FUNCTION_BLOCK PUBLIC AutomaticControl
VAR_INPUT
	Switch: BOOL;
END_VAR
VAR
	ExecutingRecipe1: BOOL := FALSE;
	ExecutingRecipe2: BOOL := FALSE;
	SwitchedManualAuto: BOOL := FALSE;
	initialized: BOOL := FALSE;
	State: INT := 0;
END_VAR
VAR_OUTPUT
	Output: BOOL;
END_VAR

// Initially go to position (0,0,0,0) and initialize motors
IF NOT IO.Initialized THEN
	Initialize();
ELSE
	//Safety();	// to stop when out of range
	
	// COUNTING (POSITION):
	CountPosition();	// FOR MANUAL MODE
	
	// RESET THE POSITION:
	(*IF (Automatic.RotationPositionAuto - Automatic.RotationPositionCurrent > 20 OR Automatic.RotationPositionAuto - Automatic.RotationPositionCurrent > 20) AND IO.SwitchedToAutomatic THEN
		IF Automatic.RotationPositionAuto - Automatic.RotationPositionCurrent > 20 THEN
			IO.MotorRotationDirection := 0;
		ELSE
			IO.MotorRotationDirection := 1;
		END_IF
		IO.MotorRotation := 1;
	ELSE 
		IO.MotorRotation := 0;
		IO.SwitchedToAutomatic := 0;
	END_IF*)
	(*IF Automatic.ExtensionPositionAuto <> Automatic.ExtensionPositionCurrent AND NOT IO.Switch THEN
		IF Automatic.ExtensionPositionAuto - Automatic.ExtensionPositionCurrent > 0 THEN
			IO.MotorExtensionDirection := 0;
		ELSE
			IO.MotorExtensionDirection := 1;
		END_IF
		IO.MotorExtension := 1;
	ELSE 
		IF NOT IO.Switch THEN
			IO.MotorExtension := 0;
		END_IF
	END_IF*)
	
	
	
	// RECIPES (recipe is sequence of moves to execute the task):
	IF ExecutingRecipe1 OR IO.ButtonUpperLeft THEN
		ExecutingRecipe1 := TRUE;
		Recipe1();
		ExecutingRecipe1 := NOT Recipe1.Ended;
	ELSIF NOT ExecutingRecipe1 AND (IO.ButtonUpperRight OR ExecutingRecipe2) THEN
		ExecutingRecipe2 := TRUE;
		Recipe2();
		ExecutingRecipe2 := NOT Recipe2.Ended;
	END_IF
	
END_IF

// for debugging purposes:
IF IO.ButtonRed THEN
	IO.Initialized := FALSE;
END_IF

RETURN;

END_FUNCTION_BLOCK

(* stored: Version 1.1.0.1, ProductVersion 3.1.4024.13
   POU AutomaticControl: Id {f9244839-88dd-4f0f-95ab-d4274120fb90}, SpecialFunc None *)
